FUNCTION Convert_REAL_TO_SINT : Hresult
VAR_INPUT
	in : REAL;
	out : REFERENCE TO SINT;
END_VAR
VAR
	converted : SINT;
END_VAR

converted := REAL_TO_SINT(in);

IF (SINT_TO_REAL(converted) <> in) THEN
	Convert_REAL_TO_SINT := INCOMPATIBLE;
	RETURN;
END_IF

out := converted;

END_FUNCTION

(* stored: Version 1.1.0.1, ProductVersion 3.1.4024.12
   POU Convert_REAL_TO_SINT: Id {a6a2f199-d202-4322-b559-ed221e03fae7}, SpecialFunc None *)
